Yaskawa INFORM job: X2_103(30,90).JBI

/JOB
//NAME X2_103(30,90)
//POS
///NPOS 434,434,434,11,0,0
///TOOL 0
///POSTYPE PULSE
///PULSE
C00000=3271,-119374,-120746,-350,28955,423
C00001=-139815,-150552,-122246,1424,14255,0
C00002=-200060,-156091,-101839,15852,59862,-55345
C00003=-224418,-53337,-27640,-2214,78542,-35069
C00004=-224438,-48029,-16239,-2251,74255,-34999
C00005=-222894,-44537,-9885,-2258,72183,-34438
C00006=-222281,-43062,-7261,-2261,71343,-34215
C00007=-219801,-41941,-6326,-2232,71409,-33379
C00008=-219801,-41166,-4818,-2238,70878,-33369
C00009=-219801,-41941,-6326,-2232,71409,-33379
C00010=-221729,-42672,-6756,-2255,71247,-34028
C00011=-221606,-41865,-5246,-2258,70739,-33978
C00012=-220679,-41360,-4730,-2248,70703,-33665
C00013=-221121,-41526,-4828,-2254,70667,-33813
C00014=-222894,-44537,-9885,-2258,72183,-34438
C00015=-224438,-48029,-16239,-2251,74255,-34999
C00016=-224391,-58970,-41460,-2187,84149,-35159
C00017=-200676,-32931,-16327,-317,66839,-14722
C00018=-188142,840,19554,1763,51642,-2042
C00019=-188000,8373,29094,1754,49640,-2018
C00020=-187946,11534,33150,1753,48768,-2011
C00021=-187952,12994,36316,1788,47570,-2035
C00022=-187946,11534,33150,1753,48768,-2011
C00023=-185876,12386,34874,-2226,48172,1956
C00024=-184694,15261,37512,-5775,48427,5518
C00025=-187925,12395,34881,1761,48145,-2013
C00026=-187893,12200,34611,1745,48210,-1998
C00027=-186938,14194,36446,1333,48088,-1587
C00028=-187893,12200,34611,1745,48210,-1998
C00029=-187946,9000,30501,1745,49095,-2005
C00030=-188087,1386,20853,1753,51122,-2028
C00031=-181732,-4900,4438,-770,58086,538
C00032=-174031,-1565,13615,-3944,54266,3743
C00033=-174319,5596,22673,-3924,52362,3698
C00034=-174429,8580,26495,-3922,51540,3684
C00035=-174433,9836,29416,-3983,50391,3728
C00036=-174429,8580,26495,-3922,51540,3684
C00037=-171116,10926,29585,-10065,52158,10061
C00038=-171940,12922,31394,-9974,52039,9961
C00039=-174482,9161,28010,-3935,50905,3687
C00040=-174468,9090,27852,-3937,50966,3690
C00041=-173667,11408,29941,-4272,50912,4030
C00042=-174468,9090,27852,-3937,50966,3690
C00043=-174358,6073,23987,-3937,51798,3704
C00044=-174072,-1158,14840,-3954,53720,3748
C00045=-173402,-7254,1011,1102,53334,3695
C00046=-173128,11811,16147,-4053,59614,3903
C00047=-173414,18752,25429,-4036,57459,3871
C00048=-173524,21666,29357,-4035,56536,3862
C00049=-173528,22669,32063,-4087,55389,3904
C00050=-173524,21666,29357,-4035,56536,3862
C00051=-172107,23003,31802,-6738,56186,6669
C00052=-172603,25249,33980,-7141,56088,7090
C00053=-173534,22315,31141,-4067,55773,3887
C00054=-175831,15088,24311,-3157,56159,2953
C00055=-175704,15840,26859,-3250,54984,3039
C00056=-174934,18176,29047,-3559,54871,3355
C00057=-175704,15840,26859,-3250,54984,3039
C00058=-175831,15088,24311,-3157,56159,2953
C00059=-173128,11811,16147,-4053,59614,3903
C00060=-158515,-47697,-14966,-51437,42315,-4350
C00061=-160188,-28820,10706,-61150,35121,-4094
C00062=-160938,-21306,18376,-62092,34254,-3699
C00063=-161219,-18227,21598,-62564,33894,-3488
C00064=-160407,-15938,23271,-62524,34443,-3379
C00065=-161219,-18227,21598,-62564,33894,-3488
C00066=-160594,-16595,22837,-62582,34299,-3378
C00067=-160592,-14820,26146,-64075,33771,-2570
C00068=-160594,-16595,22837,-62582,34299,-3378
C00069=-158698,-15537,23539,-63423,38355,-1788
C00070=-159328,-13237,25258,-63387,39000,-1639
C00071=-161141,-18339,21498,-62573,33942,-3471
C00072=-160858,-21416,18279,-62104,34303,-3680
C00073=-160103,-28926,10617,-61167,35171,-4072
C00074=-155148,-57735,-20992,-34211,37115,-7304
C00075=-144375,-92197,-43920,10369,38826,-10763
C00076=-123336,-72493,-22760,45909,48339,-7168
C00077=-110382,-36118,14049,67828,50364,-5484
C00078=-108060,-29324,20980,68768,48684,-5556
C00079=-107188,-26521,23897,69189,48032,-5626
C00080=-107504,-24071,25534,68933,48315,-5530
C00081=-107188,-26521,23897,69189,48032,-5626
C00082=-107470,-24738,25138,69020,48257,-5582
C00083=-107461,-22674,28687,69966,47830,-6220
C00084=-107470,-24738,25138,69020,48257,-5582
C00085=-107297,-26582,23837,69168,48098,-5639
C00086=-105452,-26141,24117,69389,47026,-5331
C00087=-107297,-26582,23837,69168,48098,-5639
C00088=-108171,-29382,20923,68748,48751,-5570
C00089=-110499,-36171,13998,67809,50435,-5499
C00090=-121659,-48497,-1187,64920,67113,80
C00091=-111034,-19450,-2794,41225,71575,-4827
C00092=-95590,24468,20339,13593,66440,-13992
C00093=-94636,30658,29262,13540,64031,-13917
C00094=-94266,33287,33052,13536,63014,-13897
C00095=-94260,34102,35593,13669,61899,-14031
C00096=-94266,33287,33052,13536,63014,-13897
C00097=-94257,33804,34719,13622,62273,-13984
C00098=-93260,34925,35856,13322,61987,-13631
C00099=-94257,33804,34719,13622,62273,-13984
C00100=-93131,24579,25521,13160,62983,-13463
C00101=-93277,25237,27975,13342,61865,-13653
C00102=-93655,28227,30921,13496,61658,-13825
C00103=-93277,25237,27975,13342,61865,-13653
C00104=-93131,24579,25521,13160,62983,-13463
C00105=-94266,33287,33052,13536,63014,-13897
C00106=-94636,30658,29262,13540,64031,-13917
C00107=-95590,24468,20339,13593,66440,-13992
C00108=-97908,6855,5922,13137,61050,-15522
C00109=-95297,11242,18824,14178,60690,-14590
C00110=-94266,17792,27740,14146,58451,-14474
C00111=-93867,20555,31520,14152,57502,-14440
C00112=-93860,21684,34363,14333,56366,-14591
C00113=-93867,20555,31520,14152,57502,-14440
C00114=-93834,21021,32943,14240,56879,-14511
C00115=-92751,22112,33981,13895,56618,-14106
C00116=-93834,21021,32943,14240,56879,-14511
C00117=-93847,20969,32801,14234,56940,-14507
C00118=-94233,23977,35706,14399,56772,-14687
C00119=-93847,20969,32801,14234,56940,-14507
C00120=-94245,18170,28975,14223,57899,-14539
C00121=-95277,11545,19966,14246,60155,-14652
C00122=-94527,-29265,-13111,13981,59468,-14364
C00123=-81565,-27458,3058,10852,48627,-10401
C00124=-80654,-20498,11026,10706,47205,-10165
C00125=-80308,-17644,14351,10663,46591,-10083
C00126=-80298,-16160,17342,10850,45531,-10203
C00127=-80308,-17644,14351,10663,46591,-10083
C00128=-80310,-16770,15973,10760,46052,-10147
C00129=-78983,-15416,16967,10190,45971,-9563
C00130=-80310,-16770,15973,10760,46052,-10147
C00131=-80369,-16920,15767,10776,46108,-10166
C00132=-81126,-14569,17524,11066,46330,-10477
C00133=-80369,-16920,15767,10776,46108,-10166
C00134=-80716,-19796,12409,10816,46731,-10247
C00135=-81629,-26799,4373,10955,48172,-10481
C00136=-86277,-103593,-50572,6201,53759,-1419
C00137=-92001,-164037,-66154,1441,46610,9206
C00138=-90543,-138207,-41193,1547,44504,9649
C00139=-90367,-132355,-34986,1576,43689,9693
C00140=-90296,-130023,-32460,1589,43332,9709
C00141=-104076,-127604,-31640,1030,44224,5222
C00142=-104076,-125902,-29753,1035,43937,5219
C00143=-104076,-127604,-31640,1030,44224,5222
C00144=-75365,-129597,-31294,2148,42603,14582
C00145=-79043,-127585,-29221,2027,42422,13375
C00146=-98067,-126626,-29482,1288,43342,7171
C00147=-91643,-127131,-29393,1548,42950,9262
C00148=-91643,-133346,-36144,1521,43911,9279
C00149=-90543,-138207,-41193,1547,44504,9649
C00150=-97075,-139435,-37667,8780,42441,4238
C00151=-97192,-133417,-31365,8906,41673,4121
C00152=-82208,-129108,-27879,9651,40633,8927
C00153=-74453,-129099,-27873,9918,40030,11450
C00154=-77506,-125561,-24368,25333,36038,-6444
C00155=-97622,-127372,-24807,30901,38923,-18802
C00156=-97583,-132582,-30437,30417,39596,-18508
C00157=-96835,-139510,-37769,-4213,44951,10151
C00158=-96981,-133489,-31463,-4286,44162,10144
C00159=-62865,-129479,-28052,-642,44803,20513
C00160=-78696,-129496,-28185,-2375,44685,15709
C00161=-65731,-129649,-28076,-960,44711,19643
C00162=-97517,-133431,-31347,-4343,44102,9982
C00163=-97378,-139453,-37655,-4269,44892,9987
C00164=-122537,-139380,-37444,-6562,43692,2224
C00165=-122537,-133356,-31132,-6657,42908,2284
C00166=-123909,-129354,-27957,-6756,42937,1849
C00167=-136767,-129599,-28086,-7733,42151,-2168
C00168=-136042,-129584,-28096,-7681,42205,-1941
C00169=-122565,-109770,-4675,-55538,56258,9899
C00170=-122572,-114852,-10615,-54984,56869,9434
C00171=-218346,-133610,-69952,-6045,59781,-31164
C00172=-223401,-45840,-13156,-5364,69548,-33408
C00173=-222109,-41719,-6333,-5495,67560,-32869
C00174=-220997,-38818,-2909,-5568,67023,-32457
C00175=-222242,-31345,1911,-5480,67806,-32926
C00176=-220920,-39606,-2024,-7766,59138,-23574
C00177=-220403,-51511,-7368,-9623,49930,-15864
C00178=-221089,-58034,-14727,-9279,51017,-16249
C00179=-225149,-36583,-7538,-3060,79587,-35998
C00180=-223778,-33707,-1346,-2977,77308,-35487
C00181=-222503,-31636,1503,-2884,76662,-35050
C00182=-221605,-36907,-1779,-2822,76007,-34739
C00183=-217292,-55512,-12105,-2514,72937,-33253
C00184=-219328,-56399,-14375,-2668,73818,-33940
C00185=-221046,-59770,-20585,-2780,75851,-34551
C00186=-232710,-104201,-36509,-3988,62401,-37975
C00187=-229171,-99745,-30242,-3753,60982,-36787
C00188=-225249,-97366,-27202,-3442,60481,-35515
C00189=-159716,-121406,-28671,3019,49335,-15001
C00190=-178146,-119749,-28353,3122,51852,-21289
C00191=-201053,-127933,-48461,1469,67517,-27836
C00192=-218346,-133610,-69952,-6045,59781,-31164
C00193=-155907,-158824,-62139,3482,48253,-13777
C00194=-122507,-139290,-37311,6932,43923,-3746
C00195=-122509,-133268,-31001,7032,43139,-3809
C00196=-129091,-129141,-27877,6412,43686,-5823
C00197=-103454,-129456,-28220,8487,42206,2149
C00198=-122587,-133369,-31211,7015,43220,-3827
C00199=-122586,-139389,-37517,6916,44002,-3765
C00200=-178554,-156416,-68062,-1714,49894,-19175
C00201=-213759,-120199,-38675,-7265,47820,-28777
C00202=-208805,-113975,-32275,-7533,47440,-26995
C00203=-203457,-110659,-29180,-7720,47634,-25130
C00204=-226422,-78834,-22033,-5752,57916,-33897
C00205=-229015,-79900,-24597,-5554,58778,-34856
C00206=-231182,-84689,-31124,-5352,60195,-35689
C00207=-212528,-138829,-62774,-5865,50017,-28724
C00208=-155907,-158824,-62139,3482,48253,-13777
C00209=-121094,-142626,-31574,-10098,25521,4701
C00210=-121096,-137018,-25859,-10336,24895,4818
C00211=-164582,-134101,-22446,3427,23155,-15265
C00212=-111553,-133057,-22885,-12578,25881,8893
C00213=-110779,-133123,-22850,-12777,25898,9232
C00214=-112921,-147420,-34515,-12366,25547,8360
C00215=-112921,-149481,-36511,-12292,25712,8323
C00216=-97228,-139073,-37279,8780,42400,4184
C00217=-97344,-133056,-30967,8907,41624,4066
C00218=-78012,-130084,-28544,9824,40218,10278
C00219=-81788,-129487,-28074,9683,40529,9053
C00220=-82179,-129411,-27981,9668,40535,8924
C00221=-74028,-129648,-28142,9954,39883,11573
C00222=-97200,-133072,-30998,8914,41625,4113
C00223=-97082,-139088,-37310,8787,42400,4232
C00224=-94488,-144762,-30508,4018,22458,6207
C00225=-94506,-139089,-24810,4127,21868,6148
C00226=-109156,-134471,-22107,8848,23225,-653
C00227=-92905,-135418,-22246,3518,22151,6937
C00228=-86752,-134662,-22676,6773,23151,2299
C00229=-94482,-131728,-17188,50151,23285,-24299
C00230=-94477,-136650,-22327,49039,23703,-23756
C00231=-194092,-153326,-35489,27084,38346,-44238
C00232=-219173,-157061,-72685,-6819,49419,-30815
C00233=-224435,-92754,-33276,-5864,57810,-33193
C00234=-222031,-87567,-26717,-6069,56604,-32279
C00235=-219894,-84961,-24547,-6166,56749,-31533
C00236=-220391,-83143,-23447,-6127,56973,-31723
C00237=-220808,-82168,-23250,-6081,57322,-31890
C00238=-221831,-79477,-22462,-5978,58145,-32293
C00239=-223925,-82065,-24949,-5866,58209,-33035
C00240=-226120,-87049,-31520,-5671,59544,-33877
C00241=-225186,-114904,-34894,11668,45054,-37894
C00242=-216822,-109183,-29035,10924,43485,-34913
C00243=-213756,-104039,-26334,10373,44131,-33658
C00244=-227756,-76443,-19510,10264,55464,-37669
C00245=-223895,-83934,-20074,8254,42953,-29929
C00246=-217578,-99941,-27704,3828,33118,-22325
C00247=-218675,-113856,-37596,3440,30409,-21358
C00248=-233993,-86215,-29007,10771,66078,-41518
C00249=-229810,-82565,-23340,11182,63991,-40325
C00250=-227706,-76286,-19097,11255,64337,-39587
C00251=-202149,-109903,-26387,14167,48571,-32832
C00252=-202051,-109942,-26389,14173,48540,-32803
C00253=-202051,-128717,-48625,13393,52466,-32246
C00254=-202051,-134657,-55264,13217,53473,-32112
C00255=-117234,-149912,-54866,6773,48847,-5879
C00256=-121099,-142746,-31792,-10070,25592,4686
C00257=-121100,-137139,-26082,-10306,24969,4802
C00258=-141051,-133855,-23509,-4396,24027,-4240
C00259=-121100,-133451,-23236,-10248,25112,4773
C00260=-121096,-137018,-25859,-10336,24895,4818
C00261=-121094,-142626,-31574,-10098,25521,4701
C00262=-123662,-145584,-42609,-8092,33284,3232
C00263=-230686,-106057,-33987,11415,49598,-39384
C00264=-224512,-100771,-28076,11039,47987,-37279
C00265=-205796,-94439,-26049,241,49435,-28150
C00266=-216777,-58757,-13663,-3179,61810,-31293
C00267=-233092,-64153,-16123,10229,60240,-39150
C00268=-236163,-68268,-22160,10284,62176,-40071
C00269=-236095,-83218,-48894,9648,70813,-39304
C00270=-106397,-55795,3096,63565,21817,17186
C00271=-106632,-48373,10599,65478,21584,16223
C00272=-106548,-45729,13184,65997,21437,15992
C00273=-103258,-44886,13759,64702,19643,17243
C00274=-95899,-43443,14256,59303,15873,21157
C00275=-118505,-22556,31998,69880,50592,992
C00276=-120549,-21950,32011,69247,53773,-244
C00277=-109887,-57295,-6780,52006,39852,10060
C00278=-88953,-54538,-6858,-3495,30900,36178
C00279=-87457,-47486,-1790,-16888,35291,41492
C00280=-88117,-45133,941,-16673,34715,41263
C00281=-112697,-47495,6210,47940,30588,13914
C00282=-106422,-46154,7077,44887,27834,16652
C00283=-122247,-33138,27647,79444,43496,6604
C00284=-123052,-35890,24633,78754,44065,6817
C00285=-125208,-43152,16784,77075,45600,7305
C00286=-136500,-67051,-4345,73514,52458,6539
C00287=-180716,-92339,-35753,46571,44741,-29909
C00288=-181887,-65932,-22068,22787,28646,-43428
C00289=-164154,-32069,4835,-4706,35458,-29947
C00290=-162862,-25243,12769,-5829,34168,-29145
C00291=-162318,-22407,15975,-6313,33693,-28802
C00292=-164433,-20534,17116,-4694,33821,-29993
C00293=-169618,-16577,21269,848,31718,-33215
C00294=-148668,-7920,37360,-58299,39489,-2391
C00295=-148264,-10930,34029,-57819,39984,-2589
C00296=-147210,-18873,24978,-56466,41391,-3180
C00297=-153881,-52361,-9825,-51389,40377,-7407
C00298=-195451,-44212,-13367,33096,44702,-59640
C00299=-188165,-11987,14443,28697,52592,-54038
C00300=-185681,-7933,20770,28676,50175,-53635
C00301=-185046,-6113,23212,28716,49467,-53563
C00302=-170951,-24048,16105,-1564,23385,-43494
C00303=-175189,-18557,20056,3862,23831,-46738
C00304=-164622,-16739,33688,-78292,16289,-16544
C00305=-164679,-19923,29950,-76041,16420,-17596
C00306=-165032,-27921,20991,-71332,16638,-19843
C00307=-159893,-54487,-7231,-63606,21243,-22673
C00308=-154676,-47992,-9690,-48263,49204,2905
C00309=-193585,-9261,11754,-11559,55982,16808
C00310=-194745,-2712,20199,-11444,54025,16555
C00311=-194872,621,24646,-11550,53002,16618
C00312=-184827,19619,41586,-14742,53935,20630
C00313=-184159,21046,43063,-14423,52970,15772
C00314=-184002,17429,38335,-14281,54014,15688
C00315=-182921,10224,28561,-14216,56443,15793
C00316=-177083,-111,8338,-7845,50349,39492
C00317=-178532,5317,16012,-7278,48297,39013
C00318=-179015,7475,19264,-7110,47370,38866
C00319=-178120,9780,21301,-7616,47383,39270
C00320=-171533,31347,41892,-11486,46586,42364
C00321=-173045,27120,40896,-5889,38045,43816
C00322=-172668,24060,36713,-6048,39069,43937
C00323=-171398,17656,27538,-6677,41509,44399
C00324=-161344,12362,8811,-26436,45100,67481
C00325=-163521,18252,18448,-26269,41792,67367
C00326=-161897,26643,30849,-29661,32619,71760
C00327=-161203,20965,26512,-31560,29825,74587
C00328=-161149,7456,11537,-29677,31816,73606
C00329=-175227,6351,5531,-3063,39549,38971
C00330=-186824,8866,15973,21206,34489,4565
C00331=-186762,16678,24474,21808,33336,4242
C00332=-186659,19688,27148,21766,33216,4273
C00333=-187823,20782,34277,25409,30033,2285
C00334=-189098,23597,36861,27884,33394,5871
C00335=-189065,20396,33165,27418,33944,6127
C00336=-189139,12249,23817,26457,35372,6645
C00337=-201440,-17736,15052,46372,30187,-8745
C00338=-200958,-18911,21572,51828,25568,-12457
C00339=-200198,-11285,28867,52326,24814,-12587
C00340=-199904,-8230,31793,52545,24518,-12649
C00341=-201573,-3368,42099,60720,23241,-16913
C00342=-203007,-101,44904,57709,26762,-11216
C00343=-203186,-3827,40838,56798,27185,-10789
C00344=-203962,-12064,32256,55427,28201,-10233
C00345=-200938,-30348,-961,41051,31198,-6989
C00346=-160850,-63419,-43720,34430,57956,-16775
C00347=-110095,-57810,-32372,23714,72198,-38531
C00348=-93378,-40488,-5092,23425,60303,-34603
C00349=-90533,-35882,1051,23375,58234,-33930
C00350=-89429,-33691,4119,23410,57240,-33713
C00351=-95242,-8050,22330,23694,60617,-35274
C00352=-95768,-6357,23797,23918,59729,-30488
C00353=-96526,-9092,20324,23849,60611,-30591
C00354=-98793,-14030,13298,23755,62879,-30983
C00355=-94098,-24836,421,24737,48725,-53543
C00356=-91650,-20510,6675,24341,46535,-52972
C00357=-90508,-18507,9931,24234,45316,-52749
C00358=-95414,7977,31078,26011,47297,-54577
C00359=-94573,3656,30653,27510,37763,-58721
C00360=-95383,1086,27130,27491,38776,-58811
C00361=-97471,-4004,19715,27585,41178,-59115
C00362=-94564,2818,10716,38987,45684,-75599
C00363=-92587,6675,17082,39222,43275,-75644
C00364=-91561,8164,19761,39289,42122,-75622
C00365=-92468,13395,24417,39885,42394,-76048
C00366=-93952,23755,34118,41077,42576,-76882
C00367=-90590,7329,26151,50031,24200,-87071
C00368=-96600,-9343,13340,55774,27143,-90423
C00369=-97074,-7723,20735,33897,25089,-35230
C00370=-95399,-742,27921,33089,23755,-34646
C00371=-94753,2002,30741,32759,23241,-34410
C00372=-94210,4250,38659,37485,19954,-36607
C00373=-92176,4748,39092,25289,19678,-35891
C00374=-92831,1779,35666,25549,20393,-36102
C00375=-94452,-5624,27606,26438,21912,-36738
C00376=-98858,-50483,238,51569,18835,-43949
C00377=-96204,-39490,13375,55375,15987,-45282
C00378=-95397,-37131,15438,54750,15537,-44853
C00379=-94515,-33287,24483,66247,13200,-49976
C00380=-91286,-32749,24823,46845,10625,-45650
C00381=-92274,-35440,22191,47758,11230,-46248
C00382=-94786,-42118,16150,50717,12576,-48060
C00383=-89658,-85206,-39306,19320,21137,-32731
C00384=-106882,-134348,-55470,2817,27003,-12032
C00385=-115899,-155260,-61631,-2537,28837,-4647
C00386=-121094,-142626,-31574,-10098,25521,4701
C00387=-121096,-137018,-25859,-10336,24895,4818
C00388=-164582,-134101,-22446,3427,23155,-15265
C00389=-111553,-133057,-22885,-12578,25881,8893
C00390=-110779,-133123,-22850,-12777,25898,9232
C00391=-112921,-147420,-34515,-12366,25547,8360
C00392=-112921,-149481,-36511,-12292,25712,8323
C00393=-97227,-139073,-37279,8780,42400,4185
C00394=-97341,-133056,-30967,8908,41624,4067
C00395=-78007,-130084,-28544,9824,40218,10280
C00396=-81785,-129487,-28074,9683,40529,9054
C00397=-82177,-129411,-27981,9668,40535,8924
C00398=-74024,-129648,-28142,9954,39882,11575
C00399=-97198,-133072,-30998,8914,41625,4113
C00400=-97081,-139088,-37310,8787,42400,4233
C00401=-94488,-144762,-30508,4018,22458,6207
C00402=-94506,-139089,-24810,4127,21868,6148
C00403=-109156,-134471,-22107,8848,23225,-653
C00404=-92905,-135418,-22246,3518,22151,6937
C00405=-86752,-134662,-22676,6773,23151,2299
C00406=-94482,-131728,-17188,50151,23285,-24299
C00407=-94477,-136650,-22327,49039,23703,-23756
C00408=-194092,-153326,-35489,27084,38346,-44238
C00409=-219173,-157061,-72685,-6819,49419,-30815
C00410=-224435,-92754,-33276,-5864,57810,-33193
C00411=-222031,-87567,-26717,-6069,56604,-32279
C00412=-219894,-84961,-24547,-6166,56749,-31533
C00413=-220391,-83143,-23447,-6127,56973,-31723
C00414=-220808,-82168,-23250,-6081,57322,-31890
C00415=-221831,-79477,-22462,-5978,58145,-32293
C00416=-223925,-82065,-24949,-5866,58209,-33035
C00417=-226120,-87049,-31520,-5671,59544,-33877
C00418=-225186,-114904,-34894,11668,45054,-37894
C00419=-216822,-109183,-29035,10924,43485,-34913
C00420=-213756,-104039,-26334,10373,44131,-33658
C00421=-227756,-76443,-19510,10264,55464,-37669
C00422=-223895,-83934,-20074,8254,42953,-29929
C00423=-217578,-99941,-27704,3828,33118,-22325
C00424=-218675,-113856,-37596,3440,30409,-21358
C00425=-233993,-86215,-29007,10771,66078,-41518
C00426=-229810,-82565,-23340,11182,63991,-40325
C00427=-227706,-76286,-19097,11255,64337,-39587
C00428=-202149,-109903,-26387,14167,48571,-32832
C00429=-202051,-109942,-26389,14173,48540,-32803
C00430=-202051,-128717,-48625,13393,52466,-32246
C00431=-202051,-134657,-55264,13217,53473,-32112
C00432=-134221,-121505,-102040,30238,34212,-41263
C00433=3271,-119374,-120746,-350,28955,423
BC00000=132383,666204,1075229
BC00001=261940,871255,1050994
BC00002=248524,1011966,1050994
BC00003=202466,1017054,1075175
BC00004=202466,1017054,1075175
BC00005=202466,1017054,1075175
BC00006=202466,1017054,1075175
BC00007=202466,1017054,1075175
BC00008=202466,1017054,1075175
BC00009=202466,1017054,1075175
BC00010=202466,1017054,1075175
BC00011=202466,1017054,1075175
BC00012=202466,1017054,1075175
BC00013=202466,1017054,1075175
BC00014=202466,1017054,1075175
BC00015=202466,1017054,1075175
BC00016=202466,1017054,1075175
BC00017=230796,978668,1056603
BC00018=250273,952277,1043835
BC00019=250273,952277,1043835
BC00020=250273,952277,1043835
BC00021=250273,952277,1043835
BC00022=250273,952277,1043835
BC00023=250273,952277,1043835
BC00024=250273,952277,1043832
BC00025=250273,952277,1043835
BC00026=250273,952277,1043835
BC00027=250273,952277,1043835
BC00028=250273,952277,1043835
BC00029=250273,952277,1043835
BC00030=250273,952277,1043835
BC00031=239388,961471,1057989
BC00032=226170,972635,1075175
BC00033=226170,972635,1075175
BC00034=226170,972635,1075175
BC00035=226170,972635,1075175
BC00036=226170,972635,1075175
BC00037=226170,972635,1075175
BC00038=226170,972635,1075175
BC00039=226170,972635,1075175
BC00040=226170,972635,1075175
BC00041=226170,972635,1075175
BC00042=226170,972635,1075175
BC00043=226170,972635,1075175
BC00044=226170,972635,1075175
BC00045=234013,971063,1075175
BC00046=236865,970491,1075175
BC00047=236865,970491,1075175
BC00048=236865,970491,1075175
BC00049=236865,970491,1075175
BC00050=236865,970491,1075175
BC00051=236865,970491,1075175
BC00052=236865,970491,1075175
BC00053=236865,970491,1075175
BC00054=236865,970491,1075175
BC00055=236865,970491,1075175
BC00056=236865,970491,1075175
BC00057=236865,970491,1075175
BC00058=236865,970491,1075175
BC00059=236865,970491,1075175
BC00060=241076,1045232,1015466
BC00061=241654,1055491,1007270
BC00062=241654,1055491,1007270
BC00063=241654,1055491,1007270
BC00064=241654,1055491,1007270
BC00065=241654,1055491,1007270
BC00066=241654,1055491,1007270
BC00067=241654,1055491,1007270
BC00068=241654,1055491,1007270
BC00069=241654,1055491,1007270
BC00070=241654,1055491,1007270
BC00071=241654,1055491,1007270
BC00072=241654,1055491,1007270
BC00073=241654,1055491,1007270
BC00074=243378,1058693,1018091
BC00075=246825,1065098,1039733
BC00076=250380,1071704,1062053
BC00077=248912,1056159,1048449
BC00078=248912,1056159,1048449
BC00079=248912,1056159,1048449
BC00080=248912,1056159,1048449
BC00081=248912,1056159,1048449
BC00082=248912,1056159,1048449
BC00083=248912,1056159,1048449
BC00084=248912,1056159,1048449
BC00085=248912,1056159,1048449
BC00086=248912,1056159,1048449
BC00087=248912,1056159,1048449
BC00088=248912,1056159,1048449
BC00089=248912,1056159,1048449
BC00090=248912,1056159,1060963
BC00091=253480,996710,1046754
BC00092=259276,921290,1028729
BC00093=259276,921290,1028729
BC00094=259276,921290,1028729
BC00095=259276,921290,1028729
BC00096=259276,921290,1028729
BC00097=259276,921290,1028729
BC00098=259276,921290,1028729
BC00099=259276,921290,1028729
BC00100=259276,921290,1028729
BC00101=259276,921290,1028729
BC00102=259276,921290,1028729
BC00103=259276,921290,1028729
BC00104=259276,921290,1028729
BC00105=259276,921290,1028729
BC00106=259276,921290,1028729
BC00107=259276,921290,1028729
BC00108=261148,922509,1033111
BC00109=264517,924704,1040999
BC00110=264517,924704,1040999
BC00111=264517,924704,1040999
BC00112=264517,924704,1040999
BC00113=264517,924704,1040999
BC00114=264517,924704,1040999
BC00115=264517,924704,1040999
BC00116=264517,924704,1040999
BC00117=264517,924704,1040999
BC00118=264517,924704,1040999
BC00119=264517,924704,1040999
BC00120=264517,924704,1040999
BC00121=264517,924704,1040999
BC00122=260067,934845,1062644
BC00123=257490,940717,1075175
BC00124=257490,940717,1075175
BC00125=257490,940717,1075175
BC00126=257490,940717,1075175
BC00127=257490,940717,1075175
BC00128=257490,940717,1075175
BC00129=257490,940717,1075175
BC00130=257490,940717,1075175
BC00131=257490,940717,1075175
BC00132=257490,940717,1075175
BC00133=257490,940717,1075175
BC00134=257490,940717,1075175
BC00135=257490,940717,1075175
BC00136=302625,984914,1075175
BC00137=359870,1040970,1075175
BC00138=359870,1040970,1075175
BC00139=359909,1043587,1075175
BC00140=359925,1044634,1075175
BC00141=359932,1046852,1075175
BC00142=359932,1046852,1075175
BC00143=359932,1046852,1075175
BC00144=359932,1046852,1075175
BC00145=359932,1046852,1075175
BC00146=359932,1046852,1075175
BC00147=359932,1046852,1075175
BC00148=359932,1046852,1075175
BC00149=359870,1040970,1075175
BC00150=356389,1051959,1075175
BC00151=357122,1054343,1075175
BC00152=357415,1055296,1075175
BC00153=366494,1055270,1075175
BC00154=348141,1054352,1075175
BC00155=340355,1053218,1075175
BC00156=336339,1051156,1075175
BC00157=369163,1051902,1075175
BC00158=368508,1054290,1075175
BC00159=368246,1055245,1075175
BC00160=363468,1055259,1075175
BC00161=338780,1055330,1075175
BC00162=339042,1054375,1075175
BC00163=339697,1051987,1075175
BC00164=285479,1052366,1075175
BC00165=284824,1054754,1075175
BC00166=284562,1055709,1075175
BC00167=240665,1055835,1075175
BC00168=239487,1055838,1075175
BC00169=303422,1059495,1075175
BC00170=307957,1057520,1075175
BC00171=202077,1034058,1075175
BC00172=209421,1018994,1075175
BC00173=209421,1018994,1075175
BC00174=209421,1018994,1075175
BC00175=209421,1018994,1075175
BC00176=209421,1018994,1075175
BC00177=209421,1018994,1075175
BC00178=209421,1018994,1075175
BC00179=208337,1019582,1075175
BC00180=208337,1019582,1075175
BC00181=208337,1019582,1075175
BC00182=208337,1019582,1075175
BC00183=208337,1019582,1075175
BC00184=208337,1019582,1075175
BC00185=208337,1019582,1075175
BC00186=205527,1042320,1075175
BC00187=205527,1042320,1075175
BC00188=205527,1042320,1075175
BC00189=205527,1042320,1075175
BC00190=205527,1042320,1075175
BC00191=205527,1042320,1036192
BC00192=202077,1034058,1075175
BC00193=252354,1028048,1075175
BC00194=264741,1052446,1075175
BC00195=265474,1054829,1075175
BC00196=265767,1055783,1075175
BC00197=318647,1055631,1075175
BC00198=318354,1054678,1075175
BC00199=317621,1052294,1075175
BC00200=245317,1043409,1075175
BC00201=200126,1037856,1075175
BC00202=200126,1037856,1075175
BC00203=200126,1037856,1075175
BC00204=200126,1037856,1075175
BC00205=200126,1037856,1075175
BC00206=200126,1037856,1075175
BC00207=202875,1038657,1075175
BC00208=252354,1028048,1075175
BC00209=285415,1041090,1075175
BC00210=284762,1045097,1075175
BC00211=284501,1046700,1075175
BC00212=239712,1046861,1075175
BC00213=239425,1046862,1075175
BC00214=239425,1046862,1075175
BC00215=239425,1046862,1075175
BC00216=348429,1052807,1075175
BC00217=349162,1055190,1075175
BC00218=349456,1056144,1075175
BC00219=352641,1056135,1075175
BC00220=354234,1056130,1075175
BC00221=357419,1056121,1075175
BC00222=357126,1055168,1075175
BC00223=356393,1052784,1075175
BC00224=326222,1045148,1075175
BC00225=326957,1049151,1075175
BC00226=327251,1050752,1075175
BC00227=373952,1050649,1075175
BC00228=373952,1050649,1075175
BC00229=342677,1052714,1075175
BC00230=338660,1049244,1075175
BC00231=255446,1031256,1075175
BC00232=181526,1042944,1075175
BC00233=158260,1034197,1075175
BC00234=158260,1034197,1075175
BC00235=158260,1034197,1075175
BC00236=158260,1034197,1075175
BC00237=158260,1034197,1075175
BC00238=158260,1034197,1075175
BC00239=158260,1034197,1075175
BC00240=158260,1034197,1075175
BC00241=152093,1014947,1075175
BC00242=152093,1014947,1075175
BC00243=152093,1014947,1075175
BC00244=152093,1014947,1075175
BC00245=152093,1014947,1075175
BC00246=152093,1014947,1075175
BC00247=152093,1014947,1075175
BC00248=227511,1014875,1075175
BC00249=227511,1014875,1075175
BC00250=227511,1014875,1075175
BC00251=227511,1014875,1075175
BC00252=227511,1014875,1075175
BC00253=227511,1014875,1075175
BC00254=227511,1014875,1075175
BC00255=265280,1027573,1075175
BC00256=338295,1040939,1075175
BC00257=337642,1044946,1075175
BC00258=337380,1046548,1075175
BC00259=295673,1046668,1075175
BC00260=284762,1045097,1075175
BC00261=285415,1041090,1075175
BC00262=252223,1030468,1075175
BC00263=219530,1015419,1075175
BC00264=219530,1015419,1075175
BC00265=219530,1015419,1075175
BC00266=219530,1015419,1075175
BC00267=219530,1015419,1075175
BC00268=219530,1015419,1075175
BC00269=219530,1015419,1075175
BC00270=274723,1054582,1075175
BC00271=274723,1054582,1075175
BC00272=274723,1054582,1075174
BC00273=274723,1054582,1075175
BC00274=274723,1054582,1075175
BC00275=274723,1054582,1075175
BC00276=274723,1054582,1075175
BC00277=274723,1054582,1075175
BC00278=302769,1055722,1075175
BC00279=312008,1056098,1075175
BC00280=312008,1056098,1075175
BC00281=312008,1056098,1075175
BC00282=312008,1056098,1075175
BC00283=312008,1056098,1075175
BC00284=312008,1056098,1075175
BC00285=312008,1056098,1075175
BC00286=312008,1056098,1075175
BC00287=249496,1051169,1075175
BC00288=210273,1048077,1075175
BC00289=210273,1048077,1075175
BC00290=210273,1048077,1075175
BC00291=210273,1048077,1075175
BC00292=210273,1048077,1075175
BC00293=210273,1048077,1075175
BC00294=210273,1048077,1075175
BC00295=210273,1048077,1075175
BC00296=210273,1048077,1075175
BC00297=210273,1048077,1075175
BC00298=203682,1051331,1050994
BC00299=203682,1051331,1050994
BC00300=203682,1051331,1050994
BC00301=203682,1051331,1050994
BC00302=203682,1051331,1050994
BC00303=203682,1051331,1050994
BC00304=203682,1051331,1050994
BC00305=203682,1051331,1050994
BC00306=203682,1051331,1050994
BC00307=203682,1051331,1050994
BC00308=222662,1011450,1062056
BC00309=257639,966939,1045536
BC00310=257639,966939,1045536
BC00311=257639,966939,1045536
BC00312=257639,966939,1045536
BC00313=257639,966939,1045536
BC00314=257639,966939,1045536
BC00315=257639,966939,1045536
BC00316=250000,948894,1004804
BC00317=250000,948894,1004804
BC00318=250000,948894,1004804
BC00319=250000,948894,1004804
BC00320=250000,948894,1004804
BC00321=250000,948894,1004804
BC00322=250000,948894,1004804
BC00323=250000,948894,1004804
BC00324=244323,945510,933487
BC00325=244323,945510,933487
BC00326=244323,945510,933487
BC00327=244324,945511,933483
BC00328=244324,945511,933483
BC00329=258711,950558,939336
BC00330=274206,955995,945636
BC00331=274206,955995,945636
BC00332=274206,955995,945636
BC00333=274206,955995,945636
BC00334=274206,955995,945636
BC00335=274206,955995,945636
BC00336=274206,955995,945636
BC00337=254483,964951,1031347
BC00338=249104,967393,1054722
BC00339=249104,967393,1054722
BC00340=249104,967393,1054722
BC00341=249104,967393,1054722
BC00342=249104,967393,1054722
BC00343=249104,967393,1054722
BC00344=249104,967393,1054722
BC00345=249104,967393,1054722
BC00346=260815,957267,1063697
BC00347=275794,944314,1075175
BC00348=275794,944314,1075175
BC00349=275794,944314,1075175
BC00350=275794,944314,1075175
BC00351=275794,944314,1075175
BC00352=275794,944314,1075175
BC00353=275794,944314,1075175
BC00354=275794,944314,1075175
BC00355=263746,944063,1075175
BC00356=263746,944063,1075175
BC00357=263746,944063,1075175
BC00358=263746,944063,1075175
BC00359=263746,944063,1075175
BC00360=263746,944063,1075175
BC00361=263746,944063,1075175
BC00362=235159,942078,1001811
BC00363=235159,942078,1001811
BC00364=235159,942078,1001811
BC00365=235159,942078,1001811
BC00366=235159,942078,1001811
BC00367=235159,942078,1001811
BC00368=235159,942078,1063796
BC00369=265027,925964,1060756
BC00370=265027,925964,1060756
BC00371=265027,925964,1060756
BC00372=265027,925964,1060756
BC00373=265027,925964,1060756
BC00374=265027,925964,1060756
BC00375=265027,925964,1060756
BC00376=285803,937703,1075175
BC00377=285803,937703,1075175
BC00378=285803,937703,1075175
BC00379=285803,937703,1075175
BC00380=285803,937703,1075175
BC00381=285803,937703,1075175
BC00382=285803,937703,1075175
BC00383=285803,937705,1075174
BC00384=285590,994350,1075175
BC00385=285501,1017997,1075175
BC00386=285415,1040476,1075175
BC00387=284762,1044483,1075175
BC00388=284501,1046086,1075175
BC00389=239712,1046247,1075175
BC00390=239425,1046248,1075175
BC00391=239425,1046248,1075175
BC00392=239425,1046248,1075175
BC00393=348429,1052193,1075175
BC00394=349162,1054576,1075175
BC00395=349456,1055530,1075175
BC00396=352641,1055521,1075175
BC00397=354234,1055516,1075175
BC00398=357419,1055507,1075175
BC00399=357126,1054554,1075175
BC00400=356393,1052170,1075175
BC00401=326222,1044534,1075175
BC00402=326957,1048537,1075175
BC00403=327251,1050138,1075175
BC00404=373952,1050035,1075175
BC00405=373952,1050035,1075175
BC00406=342677,1052100,1075175
BC00407=338660,1048630,1075175
BC00408=255446,1030642,1075175
BC00409=181526,1042330,1075175
BC00410=158260,1033583,1075175
BC00411=158260,1033583,1075175
BC00412=158260,1033583,1075175
BC00413=158260,1033583,1075175
BC00414=158260,1033583,1075175
BC00415=158260,1033583,1075175
BC00416=158260,1033583,1075175
BC00417=158260,1033583,1075175
BC00418=152093,1014333,1075175
BC00419=152093,1014333,1075175
BC00420=152093,1014333,1075175
BC00421=152093,1014333,1075175
BC00422=152093,1014333,1075175
BC00423=152093,1014333,1075175
BC00424=152093,1014333,1075175
BC00425=227511,1014261,1075175
BC00426=227511,1014261,1075175
BC00427=227511,1014261,1075175
BC00428=227511,1014261,1075175
BC00429=227511,1014261,1075175
BC00430=227511,1014261,1075175
BC00431=227511,1014261,1075175
BC00432=285803,876672,1075175
BC00433=132383,666204,1075229
EC00000=266052,556475
EC00001=266052,556475
EC00002=266052,556475
EC00003=266052,556475
EC00004=266052,556475
EC00005=266052,556475
EC00006=266052,556475
EC00007=266052,556475
EC00008=266052,556475
EC00009=266052,556475
EC00010=266052,556475
EC00011=266052,556475
EC00012=266052,556475
EC00013=266052,556475
EC00014=266052,556475
EC00015=266052,556475
EC00016=266052,556475
EC00017=371159,556475
EC00018=443420,556475
EC00019=443420,556475
EC00020=443420,556475
EC00021=443420,556475
EC00022=443420,556475
EC00023=443420,556475
EC00024=443419,556475
EC00025=443420,556475
EC00026=443420,556475
EC00027=443420,556475
EC00028=443420,556475
EC00029=443420,556475
EC00030=443420,556475
EC00031=443420,556475
EC00032=443420,556475
EC00033=443420,556475
EC00034=443420,556475
EC00035=443420,556475
EC00036=443420,556475
EC00037=443420,556475
EC00038=443420,556475
EC00039=443420,556475
EC00040=443420,556475
EC00041=443420,556475
EC00042=443420,556475
EC00043=443420,556475
EC00044=443420,556475
EC00045=443420,556475
EC00046=443420,556475
EC00047=443420,556475
EC00048=443420,556475
EC00049=443420,556475
EC00050=443420,556475
EC00051=443420,556475
EC00052=443420,556475
EC00053=443420,556475
EC00054=443420,556475
EC00055=443420,556475
EC00056=443420,556475
EC00057=443420,556475
EC00058=443420,556475
EC00059=443420,556475
EC00060=287458,556475
EC00061=266052,556475
EC00062=266052,556475
EC00063=266052,556475
EC00064=266052,556475
EC00065=266052,556475
EC00066=266052,556475
EC00067=266052,556475
EC00068=266052,556475
EC00069=266052,556475
EC00070=266052,556475
EC00071=266052,556475
EC00072=266052,556475
EC00073=266052,556475
EC00074=266052,556475
EC00075=266052,556475
EC00076=266052,556475
EC00077=266052,556475
EC00078=266052,556475
EC00079=266052,556475
EC00080=266052,556475
EC00081=266052,556475
EC00082=266052,556475
EC00083=266052,556475
EC00084=266052,556475
EC00085=266052,556475
EC00086=266052,556475
EC00087=266052,556475
EC00088=266052,556475
EC00089=266052,556475
EC00090=266052,556475
EC00091=344235,556475
EC00092=443420,556475
EC00093=443420,556475
EC00094=443420,556475
EC00095=443420,556475
EC00096=443420,556475
EC00097=443420,556475
EC00098=443420,556475
EC00099=443420,556475
EC00100=443420,556475
EC00101=443420,556475
EC00102=443420,556475
EC00103=443420,556475
EC00104=443420,556475
EC00105=443420,556475
EC00106=443420,556475
EC00107=443420,556475
EC00108=443420,556475
EC00109=443420,556475
EC00110=443420,556475
EC00111=443420,556475
EC00112=443420,556475
EC00113=443420,556475
EC00114=443420,556475
EC00115=443420,556475
EC00116=443420,556475
EC00117=443420,556475
EC00118=443420,556475
EC00119=443420,556475
EC00120=443420,556475
EC00121=443420,556475
EC00122=443420,556475
EC00123=443420,556475
EC00124=443420,556475
EC00125=443420,556475
EC00126=443420,556475
EC00127=443420,556475
EC00128=443420,556475
EC00129=443420,556475
EC00130=443420,556475
EC00131=443420,556475
EC00132=443420,556475
EC00133=443420,556475
EC00134=443420,556475
EC00135=443420,556475
EC00136=365225,556475
EC00137=266052,556475
EC00138=266052,556475
EC00139=266052,556475
EC00140=266052,556475
EC00141=266052,556475
EC00142=266052,556475
EC00143=266052,556475
EC00144=266052,556475
EC00145=266052,556475
EC00146=266052,556475
EC00147=266052,556475
EC00148=266052,556475
EC00149=266052,556475
EC00150=266052,556475
EC00151=266052,556475
EC00152=266052,556475
EC00153=266052,556475
EC00154=266052,556475
EC00155=266052,556475
EC00156=266052,556475
EC00157=266052,556475
EC00158=266052,556475
EC00159=266052,556475
EC00160=266052,556475
EC00161=266052,556475
EC00162=266052,556475
EC00163=266052,556475
EC00164=266052,556475
EC00165=266052,556475
EC00166=266052,556475
EC00167=266052,556475
EC00168=266052,556475
EC00169=266052,556475
EC00170=266052,556475
EC00171=266052,556475
EC00172=266052,556475
EC00173=266052,556475
EC00174=266052,556475
EC00175=266052,556475
EC00176=266052,556475
EC00177=266052,556475
EC00178=266052,556475
EC00179=266052,556475
EC00180=266052,556475
EC00181=266052,556475
EC00182=266052,556475
EC00183=266052,556475
EC00184=266052,556475
EC00185=266052,556475
EC00186=266052,556475
EC00187=266052,556475
EC00188=266052,556475
EC00189=266052,556475
EC00190=266052,556475
EC00191=266052,556475
EC00192=266052,556475
EC00193=266052,556475
EC00194=266052,556475
EC00195=266052,556475
EC00196=266052,556475
EC00197=266052,556475
EC00198=266052,556475
EC00199=266052,556475
EC00200=266052,556475
EC00201=266052,556475
EC00202=266052,556475
EC00203=266052,556475
EC00204=266052,556475
EC00205=266052,556475
EC00206=266052,556475
EC00207=266052,556475
EC00208=266052,556475
EC00209=266052,556475
EC00210=266052,556475
EC00211=266052,556475
EC00212=266052,556475
EC00213=266052,556475
EC00214=266052,556475
EC00215=266052,556475
EC00216=266052,556475
EC00217=266052,556475
EC00218=266052,556475
EC00219=266052,556475
EC00220=266052,556475
EC00221=266052,556475
EC00222=266052,556475
EC00223=266052,556475
EC00224=266052,556475
EC00225=266052,556475
EC00226=266052,556475
EC00227=266052,556475
EC00228=266052,556475
EC00229=266052,556475
EC00230=266052,556475
EC00231=266052,556475
EC00232=266052,556475
EC00233=266052,556475
EC00234=266052,556475
EC00235=266052,556475
EC00236=266052,556475
EC00237=266052,556475
EC00238=266052,556475
EC00239=266052,556475
EC00240=266052,556475
EC00241=266052,556475
EC00242=266052,556475
EC00243=266052,556475
EC00244=266052,556475
EC00245=266052,556475
EC00246=266052,556475
EC00247=266052,556475
EC00248=266052,556475
EC00249=266052,556475
EC00250=266052,556475
EC00251=266052,556475
EC00252=266052,556475
EC00253=266052,556475
EC00254=266052,556475
EC00255=266052,556475
EC00256=266052,556475
EC00257=266052,556475
EC00258=266052,556475
EC00259=266052,556475
EC00260=266052,556475
EC00261=266052,556475
EC00262=266052,556475
EC00263=266052,556475
EC00264=266052,556475
EC00265=266052,556475
EC00266=266052,556475
EC00267=266052,556475
EC00268=266052,556475
EC00269=266052,556475
EC00270=266052,556475
EC00271=266052,556475
EC00272=266052,556475
EC00273=266052,556475
EC00274=266052,556475
EC00275=266052,556475
EC00276=266052,556475
EC00277=266052,556475
EC00278=266052,556475
EC00279=266052,556475
EC00280=266052,556475
EC00281=266052,556475
EC00282=266052,556475
EC00283=266052,556475
EC00284=266052,556475
EC00285=266052,556475
EC00286=266052,556475
EC00287=266052,556475
EC00288=266052,556475
EC00289=266052,556475
EC00290=266052,556475
EC00291=266052,556475
EC00292=266052,556475
EC00293=266052,556475
EC00294=266052,556475
EC00295=266052,556475
EC00296=266052,556475
EC00297=266052,556475
EC00298=266052,556475
EC00299=266052,556475
EC00300=266052,556475
EC00301=266052,556475
EC00302=266052,556475
EC00303=266052,556475
EC00304=266052,556475
EC00305=266052,556475
EC00306=266052,556475
EC00307=266052,556475
EC00308=347188,556475
EC00309=443420,556475
EC00310=443420,556475
EC00311=443420,556475
EC00312=443420,556475
EC00313=443420,556475
EC00314=443420,556475
EC00315=443420,556475
EC00316=443420,556475
EC00317=443420,556475
EC00318=443420,556475
EC00319=443420,556475
EC00320=443420,556475
EC00321=443420,556475
EC00322=443420,556475
EC00323=443420,556475
EC00324=443420,556475
EC00325=443420,556475
EC00326=443420,556475
EC00327=443419,556475
EC00328=443419,556475
EC00329=443420,556475
EC00330=443420,556475
EC00331=443420,556475
EC00332=443420,556475
EC00333=443420,556475
EC00334=443420,556475
EC00335=443420,556475
EC00336=443420,556475
EC00337=443420,556475
EC00338=443420,556475
EC00339=443420,556475
EC00340=443420,556475
EC00341=443420,556475
EC00342=443420,556475
EC00343=443420,556475
EC00344=443420,556475
EC00345=443420,556475
EC00346=443420,556475
EC00347=443420,556475
EC00348=443420,556475
EC00349=443420,556475
EC00350=443420,556475
EC00351=443420,556475
EC00352=443420,556475
EC00353=443420,556475
EC00354=443420,556475
EC00355=443420,556475
EC00356=443420,556475
EC00357=443420,556475
EC00358=443420,556475
EC00359=443420,556475
EC00360=443420,556475
EC00361=443420,556475
EC00362=443420,556475
EC00363=443420,556475
EC00364=443420,556475
EC00365=443420,556475
EC00366=443420,556475
EC00367=443420,556475
EC00368=443420,556475
EC00369=443420,556475
EC00370=443420,556475
EC00371=443420,556475
EC00372=443420,556475
EC00373=443420,556475
EC00374=443420,556475
EC00375=443420,556475
EC00376=443420,556475
EC00377=443420,556475
EC00378=443420,556475
EC00379=443420,556475
EC00380=443420,556475
EC00381=443420,556475
EC00382=443420,556475
EC00383=443419,556475
EC00384=346238,556475
EC00385=305669,556475
EC00386=266052,556475
EC00387=266052,556475
EC00388=266052,556475
EC00389=266052,556475
EC00390=266052,556475
EC00391=266052,556475
EC00392=266052,556475
EC00393=266052,556475
EC00394=266052,556475
EC00395=266052,556475
EC00396=266052,556475
EC00397=266052,556475
EC00398=266052,556475
EC00399=266052,556475
EC00400=266052,556475
EC00401=266052,556475
EC00402=266052,556475
EC00403=266052,556475
EC00404=266052,556475
EC00405=266052,556475
EC00406=266052,556475
EC00407=266052,556475
EC00408=266052,556475
EC00409=266052,556475
EC00410=266052,556475
EC00411=266052,556475
EC00412=266052,556475
EC00413=266052,556475
EC00414=266052,556475
EC00415=266052,556475
EC00416=266052,556475
EC00417=266052,556475
EC00418=266052,556475
EC00419=266052,556475
EC00420=266052,556475
EC00421=266052,556475
EC00422=266052,556475
EC00423=266052,556475
EC00424=266052,556475
EC00425=266052,556475
EC00426=266052,556475
EC00427=266052,556475
EC00428=266052,556475
EC00429=266052,556475
EC00430=266052,556475
EC00431=266052,556475
EC00432=443420,556475
EC00433=443420,556475
///POSTYPE BASE
///RECTAN
///RCONF 0,0,0,0,0,0,0,0,0,0,0,0,0,0,0,0,0,0,0,0,0,0,0,0
P00006=0.222,-3.123,-1.508,0.0000,0.0000,0.0000
P00021=-0.225,-6.128,-0.405,0.0000,0.0000,0.0000
P00022=0.222,-3.123,-1.508,0.0000,0.0000,0.0000
P00031=1.853,-0.001,-1.549,0.0000,0.0000,0.0000
P00032=1.957,0.503,-7.217,0.0000,0.0000,0.0000
///RCONF 0,0,0,0,1,0,0,0,0,0,0,0,0,0,0,0,0,0,0,0,0,0,0,0
P00033=-0.123,0.612,-5.012,0.0000,0.0000,0.0000
///RCONF 0,0,0,0,0,0,0,0,0,0,0,0,0,0,0,0,0,0,0,0,0,0,0,0
P00034=-0.304,0.773,-2.693,0.0000,0.0000,0.0000
P00035=2.817,0.591,-1.622,0.0000,0.0000,0.0000
P00036=-1.108,-0.829,1.850,0.0000,0.0000,0.0000
P00040=-0.030,9.648,2.467,0.0000,0.0000,0.0000
P00041=0.192,3.924,0.305,0.0000,0.0000,0.0000
//INST
///DATE 2025/05/03 06:50
///ATTR SC,RW
///GROUP1 RB1,BS1
///GROUP2 ST1
NOP
'X2_103(30,90)
MOVJ C00000 BC00000 VJ=100.00  +MOVJ EC00000 VJ=100.00
MOVJ C00001 BC00001 VJ=100.00  +MOVJ EC00001 VJ=100.00
MOVJ C00002 BC00002 VJ=100.00  +MOVJ EC00002 VJ=100.00
MOVJ C00003 BC00003 VJ=15.00  +MOVJ EC00003 VJ=100.00
'Path S4757
SFTOF3D
MOVJ C00004 BC00004 VJ=100.00  +MOVJ EC00004 VJ=100.00
MOVL C00005 BC00005 V=800.0  +MOVJ EC00005 VJ=100.00
SMOVL C00006 BC00006 V=166.7  +MOVJ EC00006
SMOVL C00007 BC00007 V=166.7  +MOVJ EC00007
SREFP 3 C00008 BC00008  +REFP EC00008
CALL JOB:SEARCH-R1-S13D
SET P040 P006
SFTON3D P040
SMOVL C00009 BC00009 V=166.7  +MOVJ EC00009
SMOVL C00010 BC00010 V=166.7  +MOVJ EC00010
SMOVL C00011 BC00011 V=100.0  +MOVJ EC00011
SREFP 3 C00012 BC00012  +REFP EC00012
CALL JOB:SEARCH-R1-S13D
SET P040 P006
SFTON3D P040
SMOVL C00013 BC00013 V=166.7  +MOVJ EC00013
MOVL C00014 BC00014 V=800.0  +MOVJ EC00014 VJ=100.00
MOVL C00015 BC00015 V=1000.0  +MOVJ EC00015 VJ=100.00
'EndPath S4757
MOVJ C00016 BC00016 VJ=100.00  +MOVJ EC00016 VJ=100.00
MOVJ C00017 BC00017 VJ=100.00  +MOVJ EC00017 VJ=100.00
'Path S4795
SFTOF3D
MOVJ C00018 BC00018 VJ=100.00  +MOVJ EC00018 VJ=100.00
MOVL C00019 BC00019 V=800.0  +MOVJ EC00019 VJ=100.00
SMOVL C00020 BC00020 V=166.7  +MOVJ EC00020
SREFP 3 C00021 BC00021  +REFP EC00021
CALL JOB:SEARCH-R1-S13D
SET P031 P006
SFTON3D P031
SMOVL C00022 BC00022 V=166.7  +MOVJ EC00022
SMOVL C00023 BC00023 V=166.7  +MOVJ EC00023
SREFP 3 C00024 BC00024  +REFP EC00024
CALL JOB:SEARCH-R1-S13D
SET P031 P006
SFTON3D P031
SMOVL C00025 BC00025 V=166.7  +MOVJ EC00025
SMOVL C00026 BC00026 V=166.7  +MOVJ EC00026
SREFP 3 C00027 BC00027  +REFP EC00027
CALL JOB:SEARCH-R1-S13D
SET P031 P006
SFTON3D P031
SMOVL C00028 BC00028 V=166.7  +MOVJ EC00028
MOVL C00029 BC00029 V=800.0  +MOVJ EC00029 VJ=100.00
MOVL C00030 BC00030 V=1000.0  +MOVJ EC00030 VJ=100.00
'EndPath S4795
MOVJ C00031 BC00031 VJ=100.00  +MOVJ EC00031 VJ=100.00
'Path S4863
SFTOF3D
MOVJ C00032 BC00032 VJ=100.00  +MOVJ EC00032 VJ=100.00
MOVL C00033 BC00033 V=800.0  +MOVJ EC00033 VJ=100.00
SMOVL C00034 BC00034 V=166.7  +MOVJ EC00034
SREFP 3 C00035 BC00035  +REFP EC00035
CALL JOB:SEARCH-R1-S13D
SET P032 P006
SFTON3D P032
SMOVL C00036 BC00036 V=166.7  +MOVJ EC00036
SMOVL C00037 BC00037 V=166.7  +MOVJ EC00037
SREFP 3 C00038 BC00038  +REFP EC00038
CALL JOB:SEARCH-R1-S13D
SET P032 P006
SFTON3D P032
SMOVL C00039 BC00039 V=166.7  +MOVJ EC00039
SMOVL C00040 BC00040 V=166.7  +MOVJ EC00040
SREFP 3 C00041 BC00041  +REFP EC00041
CALL JOB:SEARCH-R1-S13D
SET P032 P006
SFTON3D P032
SMOVL C00042 BC00042 V=166.7  +MOVJ EC00042
MOVL C00043 BC00043 V=800.0  +MOVJ EC00043 VJ=100.00
MOVL C00044 BC00044 V=1000.0  +MOVJ EC00044 VJ=100.00
'EndPath S4863
MOVJ C00045 BC00045 VJ=100.00  +MOVJ EC00045 VJ=100.00
'Path S4864
SFTOF3D
MOVJ C00046 BC00046 VJ=100.00  +MOVJ EC00046 VJ=100.00
MOVL C00047 BC00047 V=800.0  +MOVJ EC00047 VJ=100.00
SMOVL C00048 BC00048 V=166.7  +MOVJ EC00048
SREFP 3 C00049 BC00049  +REFP EC00049
CALL JOB:SEARCH-R1-S13D
SET P033 P006
SFTON3D P033
SMOVL C00050 BC00050 V=166.7  +MOVJ EC00050
SMOVL C00051 BC00051 V=166.7  +MOVJ EC00051
SREFP 3 C00052 BC00052  +REFP EC00052
CALL JOB:SEARCH-R1-S13D
SET P033 P006
SFTON3D P033
SMOVL C00053 BC00053 V=166.7  +MOVJ EC00053
SMOVL C00054 BC00054 V=333.3  +MOVJ EC00054
SMOVL C00055 BC00055 V=166.7  +MOVJ EC00055
SREFP 3 C00056 BC00056  +REFP EC00056
CALL JOB:SEARCH-R1-S13D
SET P033 P006
SFTON3D P033
SMOVL C00057 BC00057 V=166.7  +MOVJ EC00057
SMOVL C00058 BC00058 V=166.7  +MOVJ EC00058
MOVL C00059 BC00059 V=1000.0  +MOVJ EC00059 VJ=100.00
'EndPath S4864
MOVJ C00060 BC00060 VJ=100.00  +MOVJ EC00060 VJ=100.00
'Path S4786
SFTOF3D
MOVJ C00061 BC00061 VJ=100.00  +MOVJ EC00061 VJ=100.00
MOVL C00062 BC00062 V=800.0  +MOVJ EC00062 VJ=100.00
SMOVL C00063 BC00063 V=166.7  +MOVJ EC00063
SREFP 3 C00064 BC00064  +REFP EC00064
CALL JOB:SEARCH-R1-S13D
SET P021 P006
SFTON3D P021
SMOVL C00065 BC00065 V=166.7  +MOVJ EC00065
SMOVL C00066 BC00066 V=166.7  +MOVJ EC00066
SREFP 3 C00067 BC00067  +REFP EC00067
CALL JOB:SEARCH-R1-S13D
SET P021 P006
SFTON3D P021
SMOVL C00068 BC00068 V=166.7  +MOVJ EC00068
SMOVL C00069 BC00069 V=166.7  +MOVJ EC00069
SREFP 3 C00070 BC00070  +REFP EC00070
CALL JOB:SEARCH-R1-S13D
SET P021 P006
SFTON3D P021
SMOVL C00071 BC00071 V=166.7  +MOVJ EC00071
MOVL C00072 BC00072 V=800.0  +MOVJ EC00072 VJ=100.00
MOVL C00073 BC00073 V=1000.0  +MOVJ EC00073 VJ=100.00
'EndPath S4786
MOVJ C00074 BC00074 VJ=100.00  +MOVJ EC00074 VJ=100.00
MOVJ C00075 BC00075 VJ=100.00  +MOVJ EC00075 VJ=100.00
MOVJ C00076 BC00076 VJ=100.00  +MOVJ EC00076 VJ=100.00
'Path S4787
SFTOF3D
MOVJ C00077 BC00077 VJ=100.00  +MOVJ EC00077 VJ=100.00
MOVL C00078 BC00078 V=800.0  +MOVJ EC00078 VJ=100.00
SMOVL C00079 BC00079 V=166.7  +MOVJ EC00079
SREFP 3 C00080 BC00080  +REFP EC00080
CALL JOB:SEARCH-R1-S13D
SET P022 P006
SFTON3D P022
SMOVL C00081 BC00081 V=166.7  +MOVJ EC00081
SMOVL C00082 BC00082 V=166.7  +MOVJ EC00082
SREFP 3 C00083 BC00083  +REFP EC00083
CALL JOB:SEARCH-R1-S13D
SET P022 P006
SFTON3D P022
SMOVL C00084 BC00084 V=166.7  +MOVJ EC00084
SMOVL C00085 BC00085 V=166.7  +MOVJ EC00085
SREFP 3 C00086 BC00086  +REFP EC00086
CALL JOB:SEARCH-R1-S13D
SET P022 P006
SFTON3D P022
SMOVL C00087 BC00087 V=166.7  +MOVJ EC00087
MOVL C00088 BC00088 V=800.0  +MOVJ EC00088 VJ=100.00
MOVL C00089 BC00089 V=1000.0  +MOVJ EC00089 VJ=100.00
'EndPath S4787
MOVJ C00090 BC00090 VJ=100.00  +MOVJ EC00090 VJ=100.00
MOVJ C00091 BC00091 VJ=100.00  +MOVJ EC00091 VJ=100.00
'Path S4800
SFTOF3D
MOVJ C00092 BC00092 VJ=100.00  +MOVJ EC00092 VJ=100.00
MOVL C00093 BC00093 V=800.0  +MOVJ EC00093 VJ=100.00
SMOVL C00094 BC00094 V=166.7  +MOVJ EC00094
SREFP 3 C00095 BC00095  +REFP EC00095
CALL JOB:SEARCH-R1-S13D
SET P036 P006
SFTON3D P036
SMOVL C00096 BC00096 V=166.7  +MOVJ EC00096
SMOVL C00097 BC00097 V=166.7  +MOVJ EC00097
SREFP 3 C00098 BC00098  +REFP EC00098
CALL JOB:SEARCH-R1-S13D
SET P036 P006
SFTON3D P036
SMOVL C00099 BC00099 V=166.7  +MOVJ EC00099
SMOVL C00100 BC00100 V=166.7  +MOVJ EC00100
SMOVL C00101 BC00101 V=166.7  +MOVJ EC00101
SREFP 3 C00102 BC00102  +REFP EC00102
CALL JOB:SEARCH-R1-S13D
SET P036 P006
SFTON3D P036
SMOVL C00103 BC00103 V=166.7  +MOVJ EC00103
SMOVL C00104 BC00104 V=166.7  +MOVJ EC00104
SMOVL C00105 BC00105 V=166.7  +MOVJ EC00105
MOVL C00106 BC00106 V=800.0  +MOVJ EC00106 VJ=100.00
MOVL C00107 BC00107 V=1000.0  +MOVJ EC00107 VJ=100.00
'EndPath S4800
MOVJ C00108 BC00108 VJ=100.00  +MOVJ EC00108 VJ=100.00
'Path S4799
SFTOF3D
MOVJ C00109 BC00109 VJ=100.00  +MOVJ EC00109 VJ=100.00
MOVL C00110 BC00110 V=800.0  +MOVJ EC00110 VJ=100.00
SMOVL C00111 BC00111 V=166.7  +MOVJ EC00111
SREFP 3 C00112 BC00112  +REFP EC00112
CALL JOB:SEARCH-R1-S13D
SET P035 P006
SFTON3D P035
SMOVL C00113 BC00113 V=166.7  +MOVJ EC00113
SMOVL C00114 BC00114 V=166.7  +MOVJ EC00114
SREFP 3 C00115 BC00115  +REFP EC00115
CALL JOB:SEARCH-R1-S13D
SET P035 P006
SFTON3D P035
SMOVL C00116 BC00116 V=166.7  +MOVJ EC00116
SMOVL C00117 BC00117 V=166.7  +MOVJ EC00117
SREFP 3 C00118 BC00118  +REFP EC00118
CALL JOB:SEARCH-R1-S13D
SET P035 P006
SFTON3D P035
SMOVL C00119 BC00119 V=166.7  +MOVJ EC00119
MOVL C00120 BC00120 V=800.0  +MOVJ EC00120 VJ=100.00
MOVL C00121 BC00121 V=1000.0  +MOVJ EC00121 VJ=100.00
'EndPath S4799
MOVJ C00122 BC00122 VJ=100.00  +MOVJ EC00122 VJ=100.00
'Path S4798
SFTOF3D
MOVJ C00123 BC00123 VJ=100.00  +MOVJ EC00123 VJ=100.00
MOVL C00124 BC00124 V=800.0  +MOVJ EC00124 VJ=100.00
SMOVL C00125 BC00125 V=166.7  +MOVJ EC00125
SREFP 3 C00126 BC00126  +REFP EC00126
CALL JOB:SEARCH-R1-S13D
SET P034 P006
SFTON3D P034
SMOVL C00127 BC00127 V=166.7  +MOVJ EC00127
SMOVL C00128 BC00128 V=166.7  +MOVJ EC00128
SREFP 3 C00129 BC00129  +REFP EC00129
CALL JOB:SEARCH-R1-S13D
SET P034 P006
SFTON3D P034
SMOVL C00130 BC00130 V=166.7  +MOVJ EC00130
SMOVL C00131 BC00131 V=166.7  +MOVJ EC00131
SREFP 3 C00132 BC00132  +REFP EC00132
CALL JOB:SEARCH-R1-S13D
SET P034 P006
SFTON3D P034
SMOVL C00133 BC00133 V=166.7  +MOVJ EC00133
MOVL C00134 BC00134 V=800.0  +MOVJ EC00134 VJ=100.00
MOVL C00135 BC00135 V=1000.0  +MOVJ EC00135 VJ=100.00
'EndPath S4798
MOVJ C00136 BC00136 VJ=100.00  +MOVJ EC00136 VJ=100.00
MOVJ C00137 BC00137 VJ=100.00  +MOVJ EC00137 VJ=100.00
'Path S4780
SFTOF3D
MOVJ C00138 BC00138 VJ=100.00  +MOVJ EC00138 VJ=100.00
MOVL C00139 BC00139 V=800.0  +MOVJ EC00139 VJ=100.00
SMOVL C00140 BC00140 V=166.7  +MOVJ EC00140
SMOVL C00141 BC00141 V=166.7  +MOVJ EC00141
SREFP 3 C00142 BC00142  +REFP EC00142
CALL JOB:SEARCH-R1-S13D
SET P041 P006
SFTON3D P041
SMOVL C00143 BC00143 V=166.7  +MOVJ EC00143
SMOVL C00144 BC00144 V=166.7  +MOVJ EC00144
SMOVL C00145 BC00145 V=100.0  +MOVJ EC00145
SREFP 3 C00146 BC00146  +REFP EC00146
CALL JOB:SEARCH-R1-S13D
SET P041 P006
SFTON3D P041
SMOVL C00147 BC00147 V=166.7  +MOVJ EC00147
SMOVL C00148 BC00148 V=250.0  +MOVJ EC00148
MOVL C00149 BC00149 V=1000.0  +MOVJ EC00149 VJ=100.00
'EndPath S4780
'Path W4762
SFTOF3D
SFTON3D P041
MOVJ C00150 BC00150 VJ=100.00  +MOVJ EC00150 VJ=100.00
SMOVL C00151 BC00151 V=800.0  +MOVJ EC00151
SMOVL C00152 BC00152 V=150.0 PL=0  +MOVJ EC00152
MACRO1 MJ#(0) ARGF9
ARCON
SMOVL C00153 BC00153 V=10.0  +MOVJ EC00153
SMOVL C00154 BC00154 V=10.0  +MOVJ EC00154
ARCOF
SMOVL C00155 BC00155 V=800.0  +MOVJ EC00155
SMOVL C00156 BC00156 V=1000.0  +MOVJ EC00156
SFTOF3D
'EndPath W4762
'Path W4764
SFTOF3D
SFTON3D P041
MOVJ C00157 BC00157 VJ=100.00  +MOVJ EC00157 VJ=100.00
SMOVL C00158 BC00158 V=800.0  +MOVJ EC00158
SMOVL C00159 BC00159 V=150.0 PL=0  +MOVJ EC00159
ARCON
SMOVL C00160 BC00160 V=10.0  +MOVJ EC00160
SMOVL C00161 BC00161 V=10.0  +MOVJ EC00161
ARCOF
SMOVL C00162 BC00162 V=800.0  +MOVJ EC00162
SMOVL C00163 BC00163 V=1000.0  +MOVJ EC00163
SFTOF3D
'EndPath W4764
'Path W4766
SFTOF3D
SFTON3D P041
MOVJ C00164 BC00164 VJ=100.00  +MOVJ EC00164 VJ=100.00
SMOVL C00165 BC00165 V=800.0  +MOVJ EC00165
SMOVL C00166 BC00166 V=150.0 PL=0  +MOVJ EC00166
ARCON
SMOVL C00167 BC00167 V=10.0  +MOVJ EC00167
SMOVL C00168 BC00168 V=10.0  +MOVJ EC00168
ARCOF
SMOVL C00169 BC00169 V=800.0  +MOVJ EC00169
SMOVL C00170 BC00170 V=1000.0  +MOVJ EC00170
SFTOF3D
'EndPath W4766
'
MOVJ C00171 BC00171 VJ=100.00  +MOVJ EC00171 VJ=100.00
'Path W4767
SFTOF3D
SFTON3D P040
MOVJ C00172 BC00172 VJ=100.00  +MOVJ EC00172 VJ=100.00
SMOVL C00173 BC00173 V=800.0  +MOVJ EC00173
SMOVL C00174 BC00174 V=150.0 PL=0  +MOVJ EC00174
ARCON
SMOVL C00175 BC00175 V=10.0  +MOVJ EC00175
SMOVL C00176 BC00176 V=10.0  +MOVJ EC00176
ARCOF
SMOVL C00177 BC00177 V=800.0  +MOVJ EC00177
SMOVL C00178 BC00178 V=1000.0  +MOVJ EC00178
SFTOF3D
'EndPath W4767
'Path W4768
SFTOF3D
SFTON3D P040
MOVJ C00179 BC00179 VJ=100.00  +MOVJ EC00179 VJ=100.00
SMOVL C00180 BC00180 V=800.0  +MOVJ EC00180
SMOVL C00181 BC00181 V=150.0 PL=0  +MOVJ EC00181
ARCON
SMOVL C00182 BC00182 V=10.0  +MOVJ EC00182
SMOVL C00183 BC00183 V=10.0  +MOVJ EC00183
ARCOF
SMOVL C00184 BC00184 V=800.0  +MOVJ EC00184
SMOVL C00185 BC00185 V=1000.0  +MOVJ EC00185
SFTOF3D
'EndPath W4768
'Path W4769
SFTOF3D
SFTON3D P040
MOVJ C00186 BC00186 VJ=100.00  +MOVJ EC00186 VJ=100.00
SMOVL C00187 BC00187 V=800.0  +MOVJ EC00187
SMOVL C00188 BC00188 V=150.0 PL=0  +MOVJ EC00188
ARCON
SMOVL C00189 BC00189 V=10.0  +MOVJ EC00189
SMOVL C00190 BC00190 V=10.0  +MOVJ EC00190
ARCOF
SMOVL C00191 BC00191 V=800.0  +MOVJ EC00191
SFTOF3D
'EndPath W4769
'
MOVJ C00192 BC00192 VJ=100.00  +MOVJ EC00192 VJ=100.00
MOVJ C00193 BC00193 VJ=100.00  +MOVJ EC00193 VJ=100.00
'Path W4765
SFTOF3D
SFTON3D P041
MOVJ C00194 BC00194 VJ=100.00  +MOVJ EC00194 VJ=100.00
SMOVL C00195 BC00195 V=800.0  +MOVJ EC00195
SMOVL C00196 BC00196 V=150.0 PL=0  +MOVJ EC00196
ARCON
SMOVL C00197 BC00197 V=10.0  +MOVJ EC00197
ARCOF
SMOVL C00198 BC00198 V=800.0  +MOVJ EC00198
SMOVL C00199 BC00199 V=1000.0  +MOVJ EC00199
SFTOF3D
'EndPath W4765
MOVJ C00200 BC00200 VJ=100.00  +MOVJ EC00200 VJ=100.00
'Path W4770
SFTOF3D
SFTON3D P040
MOVJ C00201 BC00201 VJ=100.00  +MOVJ EC00201 VJ=100.00
SMOVL C00202 BC00202 V=800.0  +MOVJ EC00202
SMOVL C00203 BC00203 V=150.0 PL=0  +MOVJ EC00203
ARCON
SMOVL C00204 BC00204 V=10.0  +MOVJ EC00204
ARCOF
SMOVL C00205 BC00205 V=800.0  +MOVJ EC00205
SMOVL C00206 BC00206 V=1000.0  +MOVJ EC00206
SFTOF3D
'EndPath W4770
MOVJ C00207 BC00207 VJ=100.00  +MOVJ EC00207 VJ=100.00
'up
MOVJ C00208 BC00208 VJ=100.00  +MOVJ EC00208 VJ=100.00
'Path W4774
SFTOF3D
SFTON3D P041
MOVJ C00209 BC00209 VJ=100.00  +MOVJ EC00209 VJ=100.00
SMOVL C00210 BC00210 V=800.0  +MOVJ EC00210
SMOVL C00211 BC00211 V=150.0 PL=0  +MOVJ EC00211
MACRO1 MJ#(0) ARGF14
ARCON
SMOVL C00212 BC00212 V=10.0  +MOVJ EC00212
SMOVL C00213 BC00213 V=10.0  +MOVJ EC00213
ARCOF
SMOVL C00214 BC00214 V=800.0  +MOVJ EC00214
SMOVL C00215 BC00215 V=1000.0  +MOVJ EC00215
SFTOF3D
'EndPath W4774
'Path W4788
SFTOF3D
SFTON3D P041
MOVJ C00216 BC00216 VJ=100.00  +MOVJ EC00216 VJ=100.00
SMOVL C00217 BC00217 V=800.0  +MOVJ EC00217
SMOVL C00218 BC00218 V=150.0 PL=0  +MOVJ EC00218
MACRO1 MJ#(0) ARGF9
ARCON
SMOVL C00219 BC00219 V=10.0  +MOVJ EC00219
SMOVL C00220 BC00220 V=10.0  +MOVJ EC00220
SMOVL C00221 BC00221 V=10.0  +MOVJ EC00221
ARCOF
SMOVL C00222 BC00222 V=800.0  +MOVJ EC00222
SMOVL C00223 BC00223 V=1000.0  +MOVJ EC00223
SFTOF3D
'EndPath W4788
'Path W4772
SFTOF3D
SFTON3D P041
MOVJ C00224 BC00224 VJ=100.00  +MOVJ EC00224 VJ=100.00
SMOVL C00225 BC00225 V=800.0  +MOVJ EC00225
SMOVL C00226 BC00226 V=150.0 PL=0  +MOVJ EC00226
MACRO1 MJ#(0) ARGF14
ARCON
SMOVL C00227 BC00227 V=10.0  +MOVJ EC00227
SMOVL C00228 BC00228 V=10.0  +MOVJ EC00228
ARCOF
SMOVL C00229 BC00229 V=800.0  +MOVJ EC00229
SMOVL C00230 BC00230 V=1000.0  +MOVJ EC00230
SFTOF3D
'EndPath W4772
MOVJ C00231 BC00231 VJ=100.00  +MOVJ EC00231 VJ=100.00
'
MOVJ C00232 BC00232 VJ=100.00  +MOVJ EC00232 VJ=100.00
'Path W4777
SFTOF3D
SFTON3D P040
MOVJ C00233 BC00233 VJ=100.00  +MOVJ EC00233 VJ=100.00
SMOVL C00234 BC00234 V=800.0  +MOVJ EC00234
SMOVL C00235 BC00235 V=150.0 PL=0  +MOVJ EC00235
MACRO1 MJ#(0) ARGF9
ARCON
SMOVL C00236 BC00236 V=10.0  +MOVJ EC00236
SMOVL C00237 BC00237 V=10.0  +MOVJ EC00237
SMOVL C00238 BC00238 V=10.0  +MOVJ EC00238
ARCOF
SMOVL C00239 BC00239 V=800.0  +MOVJ EC00239
SMOVL C00240 BC00240 V=1000.0  +MOVJ EC00240
SFTOF3D
'EndPath W4777
'Path W4778
SFTOF3D
SFTON3D P040
MOVJ C00241 BC00241 VJ=100.00  +MOVJ EC00241 VJ=100.00
SMOVL C00242 BC00242 V=800.0  +MOVJ EC00242
SMOVL C00243 BC00243 V=150.0 PL=0  +MOVJ EC00243
MACRO1 MJ#(0) ARGF14
ARCON
SMOVL C00244 BC00244 V=10.0  +MOVJ EC00244
SMOVL C00245 BC00245 V=10.0  +MOVJ EC00245
ARCOF
SMOVL C00246 BC00246 V=800.0  +MOVJ EC00246
SMOVL C00247 BC00247 V=1000.0  +MOVJ EC00247
SFTOF3D
'EndPath W4778
'Path W4776
SFTOF3D
SFTON3D P040
MOVJ C00248 BC00248 VJ=100.00  +MOVJ EC00248 VJ=100.00
SMOVL C00249 BC00249 V=800.0  +MOVJ EC00249
SMOVL C00250 BC00250 V=150.0 PL=0  +MOVJ EC00250
ARCON
SMOVL C00251 BC00251 V=10.0  +MOVJ EC00251
SMOVL C00252 BC00252 V=10.0  +MOVJ EC00252
ARCOF
SMOVL C00253 BC00253 V=800.0  +MOVJ EC00253
SMOVL C00254 BC00254 V=1000.0  +MOVJ EC00254
SFTOF3D
'EndPath W4776
'
MOVJ C00255 BC00255 VJ=100.00  +MOVJ EC00255 VJ=100.00
'Path W4773
SFTOF3D
SFTON3D P041
MOVJ C00256 BC00256 VJ=100.00  +MOVJ EC00256 VJ=100.00
SMOVL C00257 BC00257 V=800.0  +MOVJ EC00257
SMOVL C00258 BC00258 V=150.0 PL=0  +MOVJ EC00258
ARCON
SMOVL C00259 BC00259 V=9.2  +MOVJ EC00259
ARCOF
SMOVL C00260 BC00260 V=800.0  +MOVJ EC00260
SMOVL C00261 BC00261 V=1000.0  +MOVJ EC00261
SFTOF3D
'EndPath W4773
'
MOVJ C00262 BC00262 VJ=100.00  +MOVJ EC00262 VJ=100.00
'Path W4779
SFTOF3D
SFTON3D P040
MOVJ C00263 BC00263 VJ=100.00  +MOVJ EC00263 VJ=100.00
SMOVL C00264 BC00264 V=800.0  +MOVJ EC00264
SMOVL C00265 BC00265 V=150.0 PL=0  +MOVJ EC00265
ARCON
SMOVL C00266 BC00266 V=10.0  +MOVJ EC00266
ARCOF
SMOVL C00267 BC00267 V=800.0  +MOVJ EC00267
SMOVL C00268 BC00268 V=1000.0  +MOVJ EC00268
SFTOF3D
'EndPath W4779
MOVJ C00269 BC00269 VJ=100.00  +MOVJ EC00269 VJ=100.00
'
'
'
'
'uwaga na kolizje-B
'Path W4782
SFTOF3D
SFTON3D P022
MOVJ C00270 BC00270 VJ=30.00  +MOVJ EC00270 VJ=100.00
SMOVL C00271 BC00271 V=800.0  +MOVJ EC00271
'POSPAWANE
SMOVL C00272 BC00272 V=150.0 PL=0  +MOVJ EC00272
MACRO1 MJ#(0) ARGF21
ARCON
SMOVL C00273 BC00273 V=7.5  +MOVJ EC00273
SMOVL C00274 BC00274 V=7.5  +MOVJ EC00274
SMOVL C00275 BC00275 V=7.5  +MOVJ EC00275
ARCOF
SMOVL C00276 BC00276 V=800.0  +MOVJ EC00276
SMOVL C00277 BC00277 V=1000.0  +MOVJ EC00277
SFTOF3D
'Path W4789
SFTOF3D
SFTON3D P022
SMOVL C00278 BC00278 V=666.7  +MOVJ EC00278
SMOVL C00279 BC00279 V=800.0  +MOVJ EC00279
SMOVL C00280 BC00280 V=150.0 PL=0  +MOVJ EC00280
ARCON
SMOVL C00281 BC00281 V=7.5  +MOVJ EC00281
SMOVL C00282 BC00282 V=7.5  +MOVJ EC00282
SMOVL C00283 BC00283 V=7.5  +MOVJ EC00283
ARCOF
SMOVL C00284 BC00284 V=800.0  +MOVJ EC00284
SMOVL C00285 BC00285 V=1000.0  +MOVJ EC00285
SFTOF3D
'EndPath W4789
MOVJ C00286 BC00286 VJ=100.00  +MOVJ EC00286 VJ=100.00
'
MOVJ C00287 BC00287 VJ=15.00  +MOVJ EC00287 VJ=100.00
MOVJ C00288 BC00288 VJ=100.00  +MOVJ EC00288 VJ=100.00
'Path W4784
SFTOF3D
SFTON3D P021
MOVJ C00289 BC00289 VJ=100.00  +MOVJ EC00289 VJ=100.00
SMOVL C00290 BC00290 V=800.0  +MOVJ EC00290
SMOVL C00291 BC00291 V=150.0 PL=0  +MOVJ EC00291
ARCON
SMOVL C00292 BC00292 V=7.5  +MOVJ EC00292
SMOVL C00293 BC00293 V=7.5  +MOVJ EC00293
SMOVL C00294 BC00294 V=7.5  +MOVJ EC00294
ARCOF
SMOVL C00295 BC00295 V=800.0  +MOVJ EC00295
SMOVL C00296 BC00296 V=1000.0  +MOVJ EC00296
SFTOF3D
'EndPath W4784
MOVJ C00297 BC00297 VJ=100.00  +MOVJ EC00297 VJ=100.00
MOVJ C00298 BC00298 VJ=100.00  +MOVJ EC00298 VJ=100.00
'Path W4785
SFTOF3D
SFTON3D P021
MOVJ C00299 BC00299 VJ=100.00  +MOVJ EC00299 VJ=100.00
SMOVL C00300 BC00300 V=800.0  +MOVJ EC00300
SMOVL C00301 BC00301 V=150.0 PL=0  +MOVJ EC00301
ARCON
SMOVL C00302 BC00302 V=7.5  +MOVJ EC00302
SMOVL C00303 BC00303 V=7.5  +MOVJ EC00303
SMOVL C00304 BC00304 V=7.5  +MOVJ EC00304
ARCOF
SMOVL C00305 BC00305 V=800.0  +MOVJ EC00305
SMOVL C00306 BC00306 V=1000.0  +MOVJ EC00306
SFTOF3D
'EndPath W4785
MOVJ C00307 BC00307 VJ=100.00  +MOVJ EC00307 VJ=100.00
'obrot-schodki
MOVJ C00308 BC00308 VJ=100.00  +MOVJ EC00308 VJ=100.00
'Path W4790
SFTOF3D
SFTON3D P031
MOVJ C00309 BC00309 VJ=100.00  +MOVJ EC00309 VJ=100.00
SMOVL C00310 BC00310 V=800.0  +MOVJ EC00310
SMOVL C00311 BC00311 V=150.0 PL=0  +MOVJ EC00311
MACRO1 MJ#(0) ARGF9
ARCON
SMOVL C00312 BC00312 V=8.3  +MOVJ EC00312
SMOVL C00313 BC00313 V=8.3  +MOVJ EC00313
ARCOF
SMOVL C00314 BC00314 V=800.0  +MOVJ EC00314
SMOVL C00315 BC00315 V=1000.0  +MOVJ EC00315
SFTOF3D
'EndPath W4790
'Path W4865
SFTOF3D
SFTON3D P032
MOVJ C00316 BC00316 VJ=100.00  +MOVJ EC00316 VJ=100.00
SMOVL C00317 BC00317 V=800.0  +MOVJ EC00317
SMOVL C00318 BC00318 V=150.0 PL=0  +MOVJ EC00318
ARCON
SMOVL C00319 BC00319 V=8.3  +MOVJ EC00319
SMOVL C00320 BC00320 V=8.3  +MOVJ EC00320
SMOVL C00321 BC00321 V=8.3  +MOVJ EC00321
ARCOF
SMOVL C00322 BC00322 V=800.0  +MOVJ EC00322
SMOVL C00323 BC00323 V=1000.0  +MOVJ EC00323
SFTOF3D
'EndPath W4865
'Path W4866
SFTOF3D
SFTON3D P033
MOVJ C00324 BC00324 VJ=100.00  +MOVJ EC00324 VJ=100.00
SMOVL C00325 BC00325 V=150.0 PL=0  +MOVJ EC00325
ARCON
SMOVL C00326 BC00326 V=8.3  +MOVJ EC00326
ARCOF
SMOVL C00327 BC00327 V=800.0  +MOVJ EC00327
SMOVL C00328 BC00328 V=1000.0  +MOVJ EC00328
SFTOF3D
'EndPath W4866
'
MOVJ C00329 BC00329 VJ=100.00  +MOVJ EC00329 VJ=100.00
'Path W4867
SFTOF3D
SFTON3D P032
MOVJ C00330 BC00330 VJ=100.00  +MOVJ EC00330 VJ=100.00
SMOVL C00331 BC00331 V=800.0  +MOVJ EC00331
SMOVL C00332 BC00332 V=150.0 PL=0  +MOVJ EC00332
MACRO1 MJ#(0) ARGF14
ARCON
SMOVL C00333 BC00333 V=10.0  +MOVJ EC00333
SMOVL C00334 BC00334 V=10.0  +MOVJ EC00334
ARCOF
SMOVL C00335 BC00335 V=800.0  +MOVJ EC00335
SMOVL C00336 BC00336 V=1000.0  +MOVJ EC00336
SFTOF3D
'EndPath W4867
MOVJ C00337 BC00337 VJ=100.00  +MOVJ EC00337 VJ=100.00
'Path W4868
SFTOF3D
SFTON3D P031
MOVJ C00338 BC00338 VJ=100.00  +MOVJ EC00338 VJ=100.00
SMOVL C00339 BC00339 V=800.0  +MOVJ EC00339
SMOVL C00340 BC00340 V=150.0 PL=0  +MOVJ EC00340
ARCON
SMOVL C00341 BC00341 V=10.0  +MOVJ EC00341
SMOVL C00342 BC00342 V=10.0  +MOVJ EC00342
ARCOF
SMOVL C00343 BC00343 V=800.0  +MOVJ EC00343
SMOVL C00344 BC00344 V=1000.0  +MOVJ EC00344
SFTOF3D
'EndPath W4868
MOVJ C00345 BC00345 VJ=100.00  +MOVJ EC00345 VJ=100.00
'
MOVJ C00346 BC00346 VJ=100.00  +MOVJ EC00346 VJ=100.00
MOVJ C00347 BC00347 VJ=100.00  +MOVJ EC00347 VJ=100.00
'Path W4801
SFTOF3D
SFTON3D P034
MOVJ C00348 BC00348 VJ=100.00  +MOVJ EC00348 VJ=100.00
SMOVL C00349 BC00349 V=800.0  +MOVJ EC00349
SMOVL C00350 BC00350 V=150.0 PL=0  +MOVJ EC00350
MACRO1 MJ#(0) ARGF9
ARCON
SMOVL C00351 BC00351 V=8.3  +MOVJ EC00351
SMOVL C00352 BC00352 V=8.3  +MOVJ EC00352
ARCOF
SMOVL C00353 BC00353 V=800.0  +MOVJ EC00353
SMOVL C00354 BC00354 V=1000.0  +MOVJ EC00354
SFTOF3D
'EndPath W4801
'Path W4802
SFTOF3D
SFTON3D P035
MOVJ C00355 BC00355 VJ=100.00  +MOVJ EC00355 VJ=100.00
SMOVL C00356 BC00356 V=800.0  +MOVJ EC00356
SMOVL C00357 BC00357 V=150.0 PL=0  +MOVJ EC00357
ARCON
SMOVL C00358 BC00358 V=8.3  +MOVJ EC00358
SMOVL C00359 BC00359 V=8.3  +MOVJ EC00359
ARCOF
SMOVL C00360 BC00360 V=800.0  +MOVJ EC00360
SMOVL C00361 BC00361 V=1000.0  +MOVJ EC00361
SFTOF3D
'EndPath W4802
'Path W4803
SFTOF3D
SFTON3D P036
MOVJ C00362 BC00362 VJ=100.00  +MOVJ EC00362 VJ=100.00
SMOVL C00363 BC00363 V=800.0  +MOVJ EC00363
SMOVL C00364 BC00364 V=150.0 PL=0  +MOVJ EC00364
ARCON
SMOVL C00365 BC00365 V=8.3  +MOVJ EC00365
SMOVL C00366 BC00366 V=8.3  +MOVJ EC00366
ARCOF
SMOVL C00367 BC00367 V=800.0  +MOVJ EC00367
SMOVL C00368 BC00368 V=1000.0  +MOVJ EC00368
SFTOF3D
'EndPath W4803
'
'Path W4804
SFTOF3D
SFTON3D P035
MOVJ C00369 BC00369 VJ=100.00  +MOVJ EC00369 VJ=100.00
SMOVL C00370 BC00370 V=800.0  +MOVJ EC00370
SMOVL C00371 BC00371 V=150.0 PL=0  +MOVJ EC00371
MACRO1 MJ#(0) ARGF14
ARCON
SMOVL C00372 BC00372 V=10.0  +MOVJ EC00372
SMOVL C00373 BC00373 V=10.0  +MOVJ EC00373
ARCOF
SMOVL C00374 BC00374 V=800.0  +MOVJ EC00374
SMOVL C00375 BC00375 V=1000.0  +MOVJ EC00375
SFTOF3D
'EndPath W4804
'Path W4805
SFTOF3D
SFTON3D P034
MOVJ C00376 BC00376 VJ=100.00  +MOVJ EC00376 VJ=100.00
SMOVL C00377 BC00377 V=800.0  +MOVJ EC00377
SMOVL C00378 BC00378 V=150.0 PL=0  +MOVJ EC00378
ARCON
SMOVL C00379 BC00379 V=10.0  +MOVJ EC00379
SMOVL C00380 BC00380 V=10.0  +MOVJ EC00380
ARCOF
SMOVL C00381 BC00381 V=800.0  +MOVJ EC00381
SMOVL C00382 BC00382 V=1000.0  +MOVJ EC00382
SFTOF3D
COMM MOVL C00383 BC00383 V=1000.0  +MOVJ EC00383 VJ=0.78
COMM MOVL C00384 BC00384 V=1000.0  +MOVJ EC00384 VJ=0.78
COMM MOVL C00385 BC00385 V=1000.0  +MOVJ EC00385 VJ=0.78
COMM PAUSE
COMM SFTOF3D
COMM SFTON3D P041
COMM MOVJ C00386 BC00386 VJ=100.00  +MOVJ EC00386 VJ=100.00
COMM SMOVL C00387 BC00387 V=800.0  +MOVJ EC00387
COMM SMOVL C00388 BC00388 V=150.0 PL=0  +MOVJ EC00388
COMM MACRO1 MJ#(0) ARGF14
COMM ARCON
COMM SMOVL C00389 BC00389 V=13.3  +MOVJ EC00389
COMM SMOVL C00390 BC00390 V=13.3  +MOVJ EC00390
COMM ARCOF
COMM SMOVL C00391 BC00391 V=800.0  +MOVJ EC00391
COMM SMOVL C00392 BC00392 V=1000.0  +MOVJ EC00392
COMM SFTOF3D
COMM 'EndPath W4774
COMM 'Path W4788
COMM SFTOF3D
COMM SFTON3D P041
COMM MOVJ C00393 BC00393 VJ=100.00  +MOVJ EC00393 VJ=100.00
COMM SMOVL C00394 BC00394 V=800.0  +MOVJ EC00394
COMM SMOVL C00395 BC00395 V=150.0 PL=0  +MOVJ EC00395
COMM MACRO1 MJ#(0) ARGF9
COMM ARCON
COMM SMOVL C00396 BC00396 V=15.0  +MOVJ EC00396
COMM SMOVL C00397 BC00397 V=15.0  +MOVJ EC00397
COMM SMOVL C00398 BC00398 V=15.0  +MOVJ EC00398
COMM ARCOF
COMM SMOVL C00399 BC00399 V=800.0  +MOVJ EC00399
COMM SMOVL C00400 BC00400 V=1000.0  +MOVJ EC00400
COMM SFTOF3D
COMM 'EndPath W4788
COMM 'Path W4772
COMM SFTOF3D
COMM SFTON3D P041
COMM MOVJ C00401 BC00401 VJ=100.00  +MOVJ EC00401 VJ=100.00
COMM SMOVL C00402 BC00402 V=800.0  +MOVJ EC00402
COMM SMOVL C00403 BC00403 V=150.0 PL=0  +MOVJ EC00403
COMM MACRO1 MJ#(0) ARGF14
COMM ARCON
COMM SMOVL C00404 BC00404 V=15.0  +MOVJ EC00404
COMM SMOVL C00405 BC00405 V=15.0  +MOVJ EC00405
COMM ARCOF
COMM SMOVL C00406 BC00406 V=800.0  +MOVJ EC00406
COMM SMOVL C00407 BC00407 V=1000.0  +MOVJ EC00407
COMM SFTOF3D
COMM 'EndPath W4772
COMM MOVJ C00408 BC00408 VJ=100.00  +MOVJ EC00408 VJ=100.00
COMM '
COMM MOVJ C00409 BC00409 VJ=100.00  +MOVJ EC00409 VJ=100.00
COMM 'Path W4777
COMM SFTOF3D
COMM SFTON3D P040
COMM MOVJ C00410 BC00410 VJ=100.00  +MOVJ EC00410 VJ=100.00
COMM SMOVL C00411 BC00411 V=800.0  +MOVJ EC00411
COMM SMOVL C00412 BC00412 V=150.0 PL=0  +MOVJ EC00412
COMM MACRO1 MJ#(0) ARGF9
COMM ARCON
COMM SMOVL C00413 BC00413 V=13.3  +MOVJ EC00413
COMM SMOVL C00414 BC00414 V=13.3  +MOVJ EC00414
COMM SMOVL C00415 BC00415 V=13.3  +MOVJ EC00415
COMM ARCOF
COMM SMOVL C00416 BC00416 V=800.0  +MOVJ EC00416
COMM SMOVL C00417 BC00417 V=1000.0  +MOVJ EC00417
COMM SFTOF3D
COMM 'EndPath W4777
COMM 'Path W4778
COMM SFTOF3D
COMM SFTON3D P040
COMM MOVJ C00418 BC00418 VJ=100.00  +MOVJ EC00418 VJ=100.00
COMM SMOVL C00419 BC00419 V=800.0  +MOVJ EC00419
COMM SMOVL C00420 BC00420 V=150.0 PL=0  +MOVJ EC00420
COMM MACRO1 MJ#(0) ARGF14
COMM ARCON
COMM SMOVL C00421 BC00421 V=15.0  +MOVJ EC00421
COMM SMOVL C00422 BC00422 V=15.0  +MOVJ EC00422
COMM ARCOF
COMM SMOVL C00423 BC00423 V=800.0  +MOVJ EC00423
COMM SMOVL C00424 BC00424 V=1000.0  +MOVJ EC00424
COMM SFTOF3D
COMM 'EndPath W4778
COMM 'Path W4776
COMM SFTOF3D
COMM SFTON3D P040
COMM MOVJ C00425 BC00425 VJ=100.00  +MOVJ EC00425 VJ=100.00
COMM SMOVL C00426 BC00426 V=800.0  +MOVJ EC00426
COMM SMOVL C00427 BC00427 V=150.0 PL=0  +MOVJ EC00427
COMM ARCON
COMM SMOVL C00428 BC00428 V=10.0  +MOVJ EC00428
COMM SMOVL C00429 BC00429 V=10.0  +MOVJ EC00429
COMM ARCOF
COMM SMOVL C00430 BC00430 V=800.0  +MOVJ EC00430
COMM SMOVL C00431 BC00431 V=1000.0  +MOVJ EC00431
COMM SFTOF3D
COMM PAUSE
'EndPath W4805
MOVJ C00432 BC00432 VJ=100.00  +MOVJ EC00432 VJ=100.00
'
'
'
MOVJ C00433 BC00433 VJ=100.00  +MOVJ EC00433 VJ=100.00
END
